// TIA Portal V17 export
// export: Created 2023-02-25T14:41:07.0999693Z, ExportSetting WithDefaults, DisplayName Totally Integrated Automation Portal, DisplayVersion V17, DisplayName TIA Portal Openness, DisplayVersion V17, DisplayName TIA Portal Version Control Interface, DisplayVersion V17, DisplayName TIA Portal Test Suite Advanced, DisplayVersion V17, DisplayName STEP 7 Professional, DisplayVersion V17, DisplayName SIMATIC Energy Suite, DisplayVersion V17, DisplayName STEP 7 Safety, DisplayVersion V17, DisplayName WinCC Professional, DisplayVersion V17
ORGANIZATION_BLOCK "HW_Weight"   // OB30, LAD, CyclicInterrupt
{ S7_Optimized_Access := 'TRUE' }
VERSION : 0.1
// stored: AutoNumber true, IsIECCheckEnabled false, SetENOAutomatically false
   VAR_INPUT
      Initial_Call : Bool;   // Initial call of this OB
      Event_Count : Int;   // Events discarded
   END_VAR
   VAR_TEMP
      Work : Bool;
   END_VAR
   VAR_TEMP   // added for the SCL form of the ladder/FBD networks
      _w1 : Bool;
   END_VAR
BEGIN

REGION Network 1: Call: MovingAverageFilter
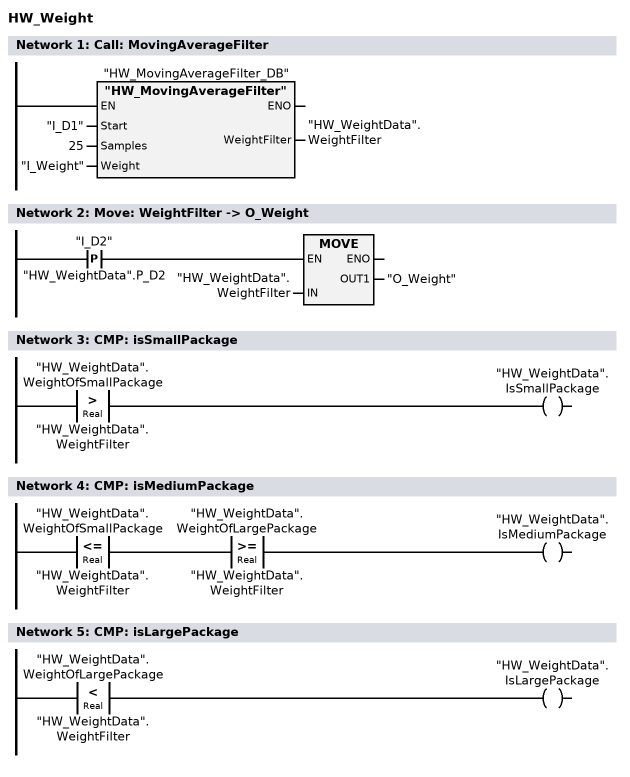
   RUNG wire#powerrail
      "HW_MovingAverageFilter_DB"(Start := "I_D1", Samples := 25, Weight := "I_Weight", WeightFilter => "HW_WeightData".WeightFilter)
   END_RUNG
   // the same network as SCL:
   "HW_MovingAverageFilter_DB"(Start := "I_D1",   // "HW_MovingAverageFilter"
                           Samples := 25,
                           Weight := "I_Weight",
                           WeightFilter => "HW_WeightData".WeightFilter);
END_REGION

REGION Network 2: Move: WeightFilter -> O_Weight
   RUNG wire#powerrail
      P_Contact(operand := "I_D2", bit := "HW_WeightData".P_D2)
      Move(in := "HW_WeightData".WeightFilter, out1 => "O_Weight")
   END_RUNG
   // the same network as SCL:
   #_w1 := "I_D2" AND NOT "HW_WeightData".P_D2;   // rising edge of "I_D2"
   "HW_WeightData".P_D2 := "I_D2";
   IF #_w1 THEN "O_Weight" := "HW_WeightData".WeightFilter; END_IF;
END_REGION

REGION Network 3: CMP: isSmallPackage
   RUNG wire#powerrail
      { S7_Templates := "SrcType := Real" } GT_Contact(in1 := "HW_WeightData".WeightOfSmallPackage, in2 := "HW_WeightData".WeightFilter)
      Coil( "HW_WeightData".IsSmallPackage )
   END_RUNG
   // the same network as SCL:
   "HW_WeightData".IsSmallPackage := "HW_WeightData".WeightOfSmallPackage > "HW_WeightData".WeightFilter;
END_REGION

REGION Network 4: CMP: isMediumPackage
   RUNG wire#powerrail
      { S7_Templates := "SrcType := Real" } LE_Contact(in1 := "HW_WeightData".WeightOfSmallPackage, in2 := "HW_WeightData".WeightFilter)
      { S7_Templates := "SrcType := Real" } GE_Contact(in1 := "HW_WeightData".WeightOfLargePackage, in2 := "HW_WeightData".WeightFilter)
      Coil( "HW_WeightData".IsMediumPackage )
   END_RUNG
   // the same network as SCL:
   "HW_WeightData".IsMediumPackage := ("HW_WeightData".WeightOfSmallPackage <= "HW_WeightData".WeightFilter) AND ("HW_WeightData".WeightOfLargePackage >= "HW_WeightData".WeightFilter);
END_REGION

REGION Network 5: CMP: isLargePackage
   RUNG wire#powerrail
      { S7_Templates := "SrcType := Real" } LT_Contact(in1 := "HW_WeightData".WeightOfLargePackage, in2 := "HW_WeightData".WeightFilter)
      Coil( "HW_WeightData".IsLargePackage )
   END_RUNG
   // the same network as SCL:
   "HW_WeightData".IsLargePackage := "HW_WeightData".WeightOfLargePackage < "HW_WeightData".WeightFilter;
END_REGION
END_ORGANIZATION_BLOCK
